FUNCTION_BLOCK Test_TEvent_AddHandlerAddsHandlerToEventHandlerList EXTENDS TUnitTestBase
VAR
    TestEvent : TTestEvent;
    TestEventHandler : TTestEventHandler;
END_VAR

TestEvent
    .ClearEventHandlers()
    .AddEventHandler(TestEventHandler);
    
Assertion.AssertEquals_UDINT(
    Expected      := 1,
    Actual        := TestEvent.EventHandlers.Count,
    VariableName  := 'TestEvent.EventHandlers.Count');
    

_TestFinished := TRUE;

END_FUNCTION_BLOCK

(* stored: Version 1.1.0.1, ProductVersion 3.1.4024.4
   POU Test_TEvent_AddHandlerAddsHandlerToEventHandlerList: Id {efe09656-7795-4a2e-b669-dba8c20969d5}, SpecialFunc None *)
